// TIA Portal V20 export
FUNCTION "07 T10 LANT LEV2" : Void   // FC1793, LAD
TITLE = TRACKING - LEV2
{ S7_Optimized_Access := 'TRUE' }
// stored: AutoNumber false, SetENOAutomatically false
   VAR_TEMP
      "HSK Answer OK" : Bool;
      Trc_OK : Bool;
      Aux_Int : Int;
      Aux_Bool : Bool;
   END_VAR
BEGIN

REGION Network 1: ============ Manual movement ============
END_REGION

REGION Network 2: ============ Handshake mamnagement ============
END_REGION

REGION Network 3: Check OK / not OK
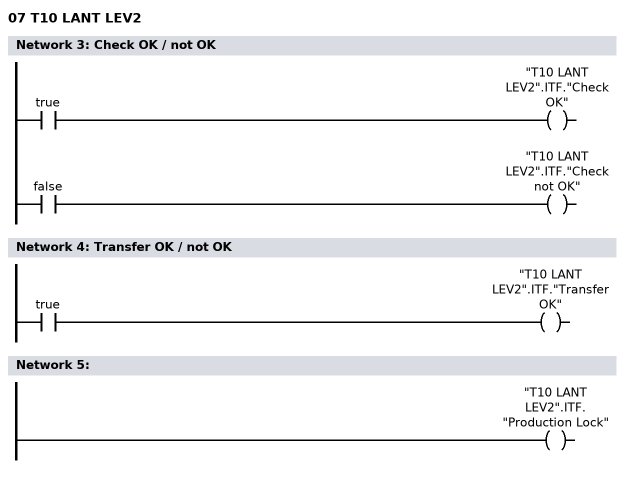
   RUNG wire#powerrail
      Contact( true )
      Coil( "T10 LANT LEV2".ITF."Check OK" )
   END_RUNG
   RUNG wire#powerrail
      Contact( false )
      Coil( "T10 LANT LEV2".ITF."Check not OK" )
   END_RUNG
   // the same network as SCL:
   "T10 LANT LEV2".ITF."Check OK" := true;
   "T10 LANT LEV2".ITF."Check not OK" := false;
END_REGION

REGION Network 4: Transfer OK / not OK
   RUNG wire#powerrail
      Contact( true )
      Coil( "T10 LANT LEV2".ITF."Transfer OK" )
   END_RUNG
   // the same network as SCL:
   "T10 LANT LEV2".ITF."Transfer OK" := true;
END_REGION

REGION Network 5
   RUNG wire#powerrail
      Coil( "T10 LANT LEV2".ITF."Production Lock" )
   END_RUNG
   // the same network as SCL:
   "T10 LANT LEV2".ITF."Production Lock" := TRUE;
END_REGION
END_FUNCTION
